SUBAPPLICATION Uebung_014 (* Subapplication Type *)
  (* Standard: 61499-2 *)
  (* Version 1.0, 2023-10-23, franz *)
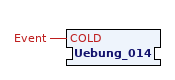
  EVENT_INPUT
    COLD;
  END_EVENT
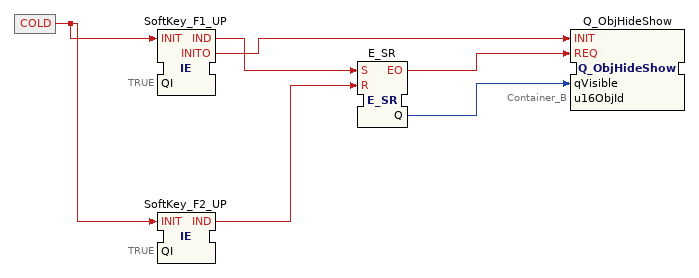
  FBS
    SoftKey_F1_UP : IE(QI := TRUE);
    SoftKey_F2_UP : IE(QI := TRUE);
    E_SR : E_SR;
    Q_ObjHideShow : Q_ObjHideShow(u16ObjId := Container_B);
  END_FBS
  EVENT_CONNECTIONS
    COLD TO SoftKey_F1_UP.INIT;
    COLD TO SoftKey_F2_UP.INIT;
    SoftKey_F1_UP.IND TO E_SR.S;
    SoftKey_F2_UP.IND TO E_SR.R;
    SoftKey_F1_UP.INITO TO Q_ObjHideShow.INIT;
    E_SR.EO TO Q_ObjHideShow.REQ;
  END_CONNECTIONS
  DATA_CONNECTIONS
    E_SR.Q TO Q_ObjHideShow.qVisible;
  END_CONNECTIONS
END_SUBAPPLICATION
